PROGRAM MAIN
VAR
	TabletFillingControl01	: 	TabletFillingControl01;
	TabletFillingControl02	: 	TabletFillingControl02;
END_VAR

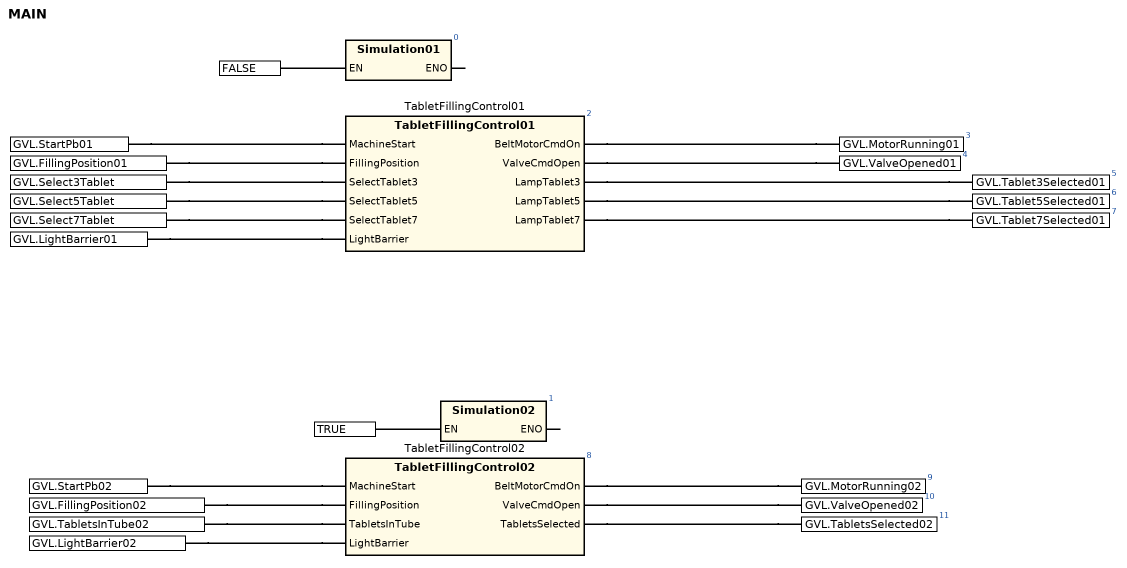
IF FALSE THEN Simulation01(); END_IF
Simulation02();
TabletFillingControl01(
    MachineStart := GVL.StartPb01,
    FillingPosition := GVL.FillingPosition01,
    SelectTablet3 := GVL.Select3Tablet,
    SelectTablet5 := GVL.Select5Tablet,
    SelectTablet7 := GVL.Select7Tablet,
    LightBarrier := GVL.LightBarrier01);
GVL.MotorRunning01 := TabletFillingControl01.BeltMotorCmdOn;
GVL.ValveOpened01 := TabletFillingControl01.ValveCmdOpen;
GVL.Tablet3Selected01 := TabletFillingControl01.LampTablet3;
GVL.Tablet5Selected01 := TabletFillingControl01.LampTablet5;
GVL.Tablet7Selected01 := TabletFillingControl01.LampTablet7;
TabletFillingControl02(
    MachineStart := GVL.StartPb02,
    FillingPosition := GVL.FillingPosition02,
    TabletsInTube := GVL.TabletsInTube02,
    LightBarrier := GVL.LightBarrier02);
GVL.MotorRunning02 := TabletFillingControl02.BeltMotorCmdOn;
GVL.ValveOpened02 := TabletFillingControl02.ValveCmdOpen;
GVL.TabletsSelected02 := TabletFillingControl02.TabletsSelected;

END_PROGRAM

(* stored: Version 1.1.0.1, ProductVersion 3.1.4024.15
   POU MAIN: Id {125b7c6e-403b-474f-807e-e894751bcd97}, SpecialFunc None *)
